PROGRAM INTERNAL PRG_TESTS

(* Instantiate test suites here. Naming convention for tests should be a suffix with _Tests.
Good practice for creating test methods is to end them with _test as well. *)
VAR
	AdsHelperTests					: FB_AdsHelper_Tests;
	ArrayHelperTests				: FB_ArrayHelper_Tests;
	DateTimeToStringConverterTest	: FB_DateTimeToStringConverter_Tests;
	ErrorSourceTests				: FB_ErrorSource_Tests;
	HasInstanceNameTests			: FB_HasInstanceName_Tests;
	StringBuilderTests				: FB_StringBuilder_Tests;
	HasTaskInfoTests				: FB_HasTaskInfo_Tests;
	BoolExTests						: FB_BoolEx_Tests;
	EthercatHelperTests				: FB_EthercatHelper_Tests;
	//EthercatDiagnosisTests			: FB_EthercatDiagnosis_Tests;
	MallocTests						: FB_Malloc_Tests;
	StringHelperTests				: FB_StringHelper_Tests;
	LocalSystemTimeTests			: FB_LocalSystemTime_Tests;
END_VAR

// Run tests in paralel
//TcUnit.RUN();

// Run tests in sequence, one after the other. Uncomment if required.
TcUnit.RUN_IN_SEQUENCE();

END_PROGRAM

(* stored: Version 1.1.0.1, ProductVersion 3.1.4024.15
   POU PRG_TESTS: Id {dcd11036-52e9-4f92-9371-f8c187305968}, SpecialFunc None *)
